Fanuc KAREL source: compact_preamble.KL

PROGRAM NC0001
%NOLOCKGROUP
ROUTINE R
VAR
S1:INTEGER
BEGIN
S1=1
S1=(S1 + 1)
END R
BEGIN
R
END NC0001
